{attribute 'GeneratedUsingTerminal: EL3602-0002-0016'}
{attribute addProperty BoxType "EL3602-0002-0016"}
{attribute addProperty Id "StatusAT %I*Status_F2CE6D917ValueAT %I*DINT4"}
{attribute addProperty CRC "1159803140"}
{attribute addProperty Size "11"}
TYPE AI_Inputs_Channel_45213104 EXTENDS InputBase_8311D824 :
STRUCT
	{attribute addProperty Name "Status"}
	Status AT %I* : Status_F2CE6D91;
	{attribute addProperty Name "Value"}
	Value AT %I* : DINT;
END_STRUCT
END_TYPE

(* stored: Version 1.2.0.0, ProductVersion 3.1.4024.9
   DUT AI_Inputs_Channel_45213104: Id {e873c6e8-0374-4a46-9455-1716a7022cef} *)
